% RSLogix 500 project I2P-JOB13-ADAM BOCZKIEWICZ_BAK018.RSS, saved by version 10.00.00.00 %
PROJECT "ML04A"    % processor: Bul.1763 MicroLogix 1100 Series B %

PROGRAM FILES
  LAD 2   8 rungs

DATA FILES
  O0 OUTPUT  4 elements
  I1 INPUT  6 elements
  S2 STATUS  66 elements
  B3 BINARY  1 elements
  T4 TIMER  1 elements
  C5 COUNTER  1 elements
  R6 CONTROL  1 elements
  N7 INTEGER  1 elements
  F8 FLOAT  1 elements

LADDER 2
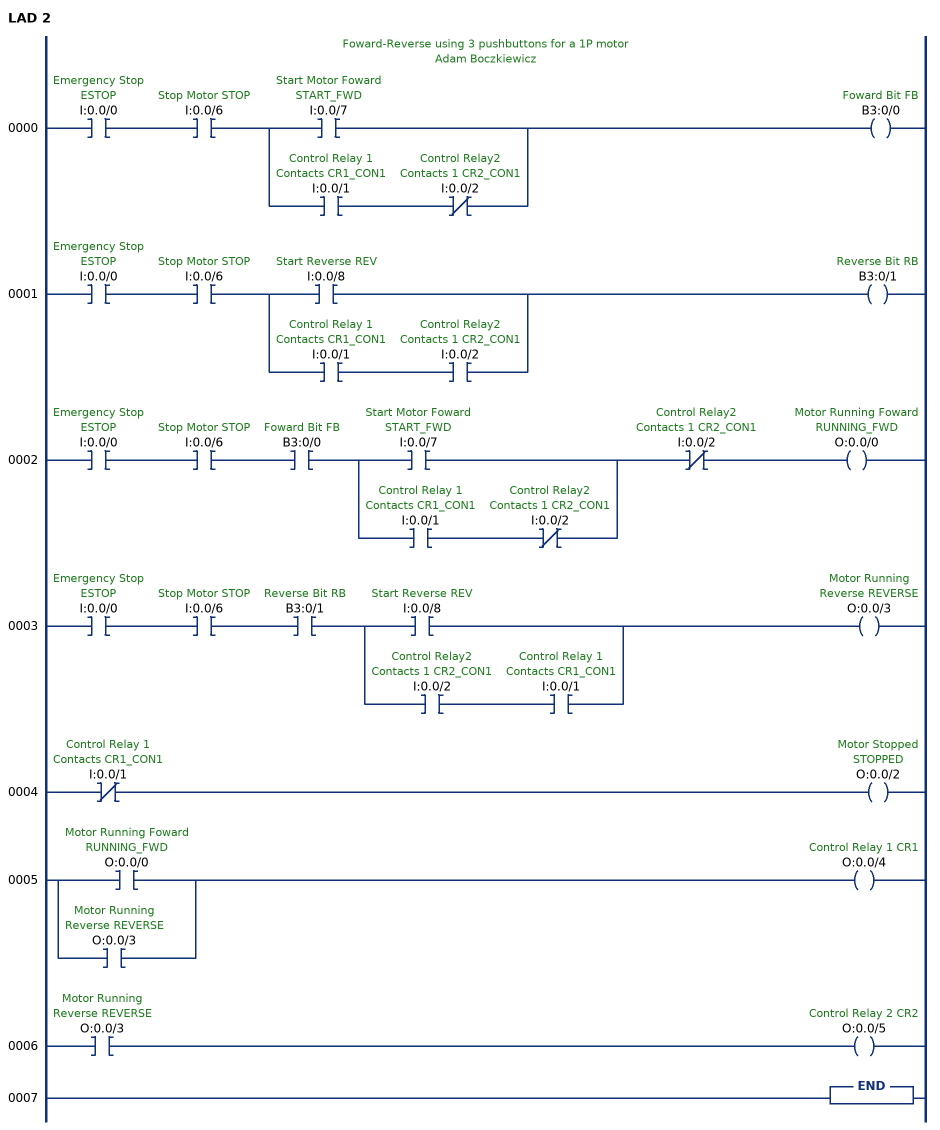
% Rung: 0 %
% Foward-Reverse using 3 pushbuttons for a 1P motor
% Adam Boczkiewicz %
SOR XIC I:0.0/0 XIC I:0.0/6 BST XIC I:0.0/7 NXB XIC I:0.0/1 XIO I:0.0/2 BND OTE B3:0/0 EOR
%   I:0.0/0  ESTOP  "Emergency Stop" %
%   I:0.0/6  STOP  "Stop Motor" %
%   I:0.0/7  START_FWD  "Start Motor Foward" %
%   I:0.0/1  CR1_CON1  "Control Relay 1 Contacts" %
%   I:0.0/2  CR2_CON1  "Control Relay2 Contacts 1" %
%   B3:0/0  FB  "Foward Bit" %
% Rung: 1 %
SOR XIC I:0.0/0 XIC I:0.0/6 BST XIC I:0.0/8 NXB XIC I:0.0/1 XIC I:0.0/2 BND OTE B3:0/1 EOR
%   I:0.0/0  ESTOP  "Emergency Stop" %
%   I:0.0/6  STOP  "Stop Motor" %
%   I:0.0/8  REV  "Start Reverse" %
%   I:0.0/1  CR1_CON1  "Control Relay 1 Contacts" %
%   I:0.0/2  CR2_CON1  "Control Relay2 Contacts 1" %
%   B3:0/1  RB  "Reverse Bit" %
% Rung: 2 %
SOR XIC I:0.0/0 XIC I:0.0/6 XIC B3:0/0 BST XIC I:0.0/7 NXB XIC I:0.0/1 XIO I:0.0/2 BND XIO I:0.0/2 OTE O:0.0/0 EOR
%   I:0.0/0  ESTOP  "Emergency Stop" %
%   I:0.0/6  STOP  "Stop Motor" %
%   B3:0/0  FB  "Foward Bit" %
%   I:0.0/7  START_FWD  "Start Motor Foward" %
%   I:0.0/1  CR1_CON1  "Control Relay 1 Contacts" %
%   I:0.0/2  CR2_CON1  "Control Relay2 Contacts 1" %
%   O:0.0/0  RUNNING_FWD  "Motor Running Foward" %
% Rung: 3 %
SOR XIC I:0.0/0 XIC I:0.0/6 XIC B3:0/1 BST XIC I:0.0/8 NXB XIC I:0.0/2 XIC I:0.0/1 BND OTE O:0.0/3 EOR
%   I:0.0/0  ESTOP  "Emergency Stop" %
%   I:0.0/6  STOP  "Stop Motor" %
%   B3:0/1  RB  "Reverse Bit" %
%   I:0.0/8  REV  "Start Reverse" %
%   I:0.0/2  CR2_CON1  "Control Relay2 Contacts 1" %
%   I:0.0/1  CR1_CON1  "Control Relay 1 Contacts" %
%   O:0.0/3  REVERSE  "Motor Running Reverse" %
% Rung: 4 %
SOR XIO I:0.0/1 OTE O:0.0/2 EOR
%   I:0.0/1  CR1_CON1  "Control Relay 1 Contacts" %
%   O:0.0/2  STOPPED  "Motor Stopped" %
% Rung: 5 %
SOR BST XIC O:0.0/0 NXB XIC O:0.0/3 BND OTE O:0.0/4 EOR
%   O:0.0/0  RUNNING_FWD  "Motor Running Foward" %
%   O:0.0/3  REVERSE  "Motor Running Reverse" %
%   O:0.0/4  CR1  "Control Relay 1" %
% Rung: 6 %
SOR XIC O:0.0/3 OTE O:0.0/5 EOR
%   O:0.0/3  REVERSE  "Motor Running Reverse" %
%   O:0.0/5  CR2  "Control Relay 2" %
% Rung: 7 %
SOR END EOR

OTHER DOCUMENTED ADDRESSES
  I:0.0/3  DIRECTION  "Direction:Forward- off-reverse"
  I:0.0/4  DIRECTION_  "Direction: Forward- Off-Reverse"
  I:0.0/5  2PSS  "2 Position Selector Switch"
  O:0.0/1  YL  "Yellow light"
